FUNCTION_BLOCK IA_WBSD (* ISOBUS Adapter for Wheel Based Speed and Distance (WBSD) *)
  (* Standard: ISO 11783-7; Classification: PGN 65096; Description: Copyright (c) 2024 HR Agrartechnik GmbH This program and the accompanying materials are made available under the terms of the Eclipse Public License 2.0 which is available at https://www.eclipse.org/legal/epl-2.0/ SPDX-License-Identifier: EPL-2.0 *)
  (* Version 1.1, 2026-04-19, Franz Höpfinger, HR Agrartechnik GmbH, Fixed: Use conversion blocks to properly connect internal pins to adapter plugs *)
  (* Version 1.0, 2026-04-19, Franz Höpfinger, HR Agrartechnik GmbH, initial API and implementation (Adapter Wrapper for I_WBSD) *)
  PACKAGE isobus::tecu;
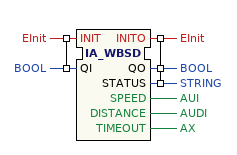
  EVENT_INPUT
    INIT : EInit WITH QI; (* Service Initialization *)
  END_EVENT
  EVENT_OUTPUT
    INITO : EInit WITH QO, STATUS; (* Initialization Confirm *)
  END_EVENT
  VAR_INPUT
    QI : BOOL; (* Event Input Qualifier *)
  END_VAR
  VAR_OUTPUT
    QO : BOOL; (* Event Output Qualifier *)
    STATUS : STRING;
  END_VAR
  PLUGS
    SPEED : adapter::types::unidirectional::AUI; (* Wheel-based machine speed *)
    DISTANCE : adapter::types::unidirectional::AUDI; (* Wheel-based machine distance *)
    TIMEOUT : adapter::types::unidirectional::AX; (* Timeout Status *)
  END_PLUGS
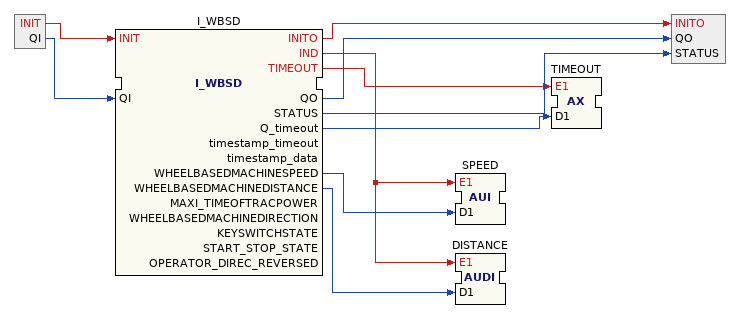
  FBS
    I_WBSD : isobus::tecu::I_WBSD;
  END_FBS
  EVENT_CONNECTIONS
    INIT TO I_WBSD.INIT;
    I_WBSD.INITO TO INITO;
    I_WBSD.TIMEOUT TO TIMEOUT.E1;
    I_WBSD.IND TO DISTANCE.E1;
    I_WBSD.IND TO SPEED.E1;
  END_CONNECTIONS
  DATA_CONNECTIONS
    QI TO I_WBSD.QI;
    I_WBSD.QO TO QO;
    I_WBSD.STATUS TO STATUS;
    I_WBSD.Q_timeout TO TIMEOUT.D1;
    I_WBSD.WHEELBASEDMACHINESPEED TO SPEED.D1;
    I_WBSD.WHEELBASEDMACHINEDISTANCE TO DISTANCE.D1;
  END_CONNECTIONS
END_FUNCTION_BLOCK
